Staubli VAL3: saveTool.pjx

--- saveTool.pjx ---
Parameters version=s7.2.1 stackSize=5000 millimeterUnit=true
Data file=saveTool.dtx
Library alias=io path=Disk://io/io.pjx

--- saveTool.dtx ---
public string name[2]
public string sActionOFF[2]
  [0] = "CALL OFF^^"
  [1] = "CALL OFF^^"
public string sActionON[2]
  [0] = "CALL ON^^"
  [1] = "CALL ON^^"
public bool bCheck = true
public pointRx rif2 = {x=987.30721, y=10.835485, z=1375.350782, rx=1.315674, ry=-0.828127, rz=-86.484115, shoulder=lefty, elbow=enegative, wrist=wpositive, fatherId=world[0]}
public mdesc nom_speed = {rmax=9999, blend=off}
public tool gun[2]
  [0] = {x=-234.5, y=4.7, z=169.7, ry=-90, fatherId=flange[0], ioLink=valve1}
  [1] = {x=-234.5, y=4.7, z=169.7, ry=-90, fatherId=flange[0], ioLink=valve1}
